(* PLC project Unnamed, Unknown Unnamed 1 *)
(* stored: creationDateTime 2026-08-16T23:05:33, modificationDateTime 2026-08-16T23:05:33 *)

FUNCTION_BLOCK CTU
  VAR_OUTPUT
    Q : BOOL;
    CV : INT;
  END_VAR
  VAR_INPUT
    CU : BOOL;
    R : BOOL;
    PV : INT;
  END_VAR

END_FUNCTION_BLOCK

FUNCTION_BLOCK F_TRIG
  VAR_OUTPUT
    Q : BOOL;
  END_VAR
  VAR_INPUT
    CLK : BOOL;
  END_VAR

END_FUNCTION_BLOCK

FUNCTION_BLOCK R_TRIG
  VAR_OUTPUT
    Q : BOOL;
  END_VAR
  VAR_INPUT
    CLK : BOOL;
  END_VAR

END_FUNCTION_BLOCK

FUNCTION_BLOCK SR
  VAR_OUTPUT
    Q1 : BOOL;
  END_VAR
  VAR_INPUT
    S1 : BOOL;
    R : BOOL;
  END_VAR

END_FUNCTION_BLOCK

FUNCTION_BLOCK TON
  VAR_OUTPUT
    Q : BOOL;
    ET : TIME;
  END_VAR
  VAR_INPUT
    IN : BOOL;
    PT : TIME;
  END_VAR

END_FUNCTION_BLOCK

PROGRAM main
  VAR
    Start_PB AT %QX1.0 : BOOL;  (* Simulated pushbutton, driven externally via Modbus coil *)
    Stop_PB AT %QX1.1 : BOOL;
    EStop_OK AT %QX1.2 : BOOL;
    Jam_Sensor AT %QX1.3 : BOOL;
    Part_Present AT %QX1.4 : BOOL;
    Reject_Sensor AT %QX1.5 : BOOL;
    Reset_PB AT %QX1.6 : BOOL;
    Conveyor_Motor AT %QX0.3 : BOOL;
    Fill_Actuator AT %QX0.4 : BOOL;
    Fault_Lamp AT %QX0.5 : BOOL;
    Reject_Gate AT %QX0.2 : BOOL;
    Machine_Running AT %QX0.0 : BOOL;
    Machine_Faulted AT %QX0.1 : BOOL;
    Cycle_Count AT %MW0 : INT;
    Good_Count AT %MW1 : INT;
    Reject_Count AT %MW2 : INT;
  END_VAR
  VAR
    SR0 : SR;
    R_TRIG0 : R_TRIG;
    Part_Edge : BOOL;
    CTU0 : CTU;
    TON0 : TON;
    CTU1 : CTU;
    CTU2 : CTU;
    TON1 : TON;
    F_TRIG0 : F_TRIG;
    Fault_Cleared : BOOL;
  END_VAR

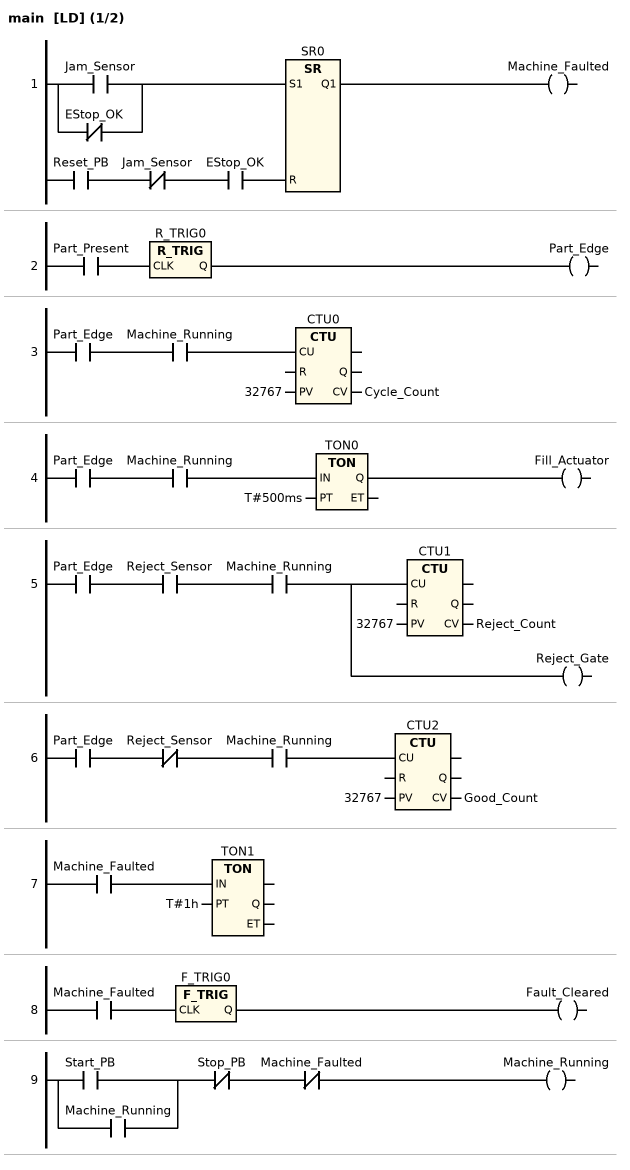
(* LD diagram, written out as Structured Text *)
Machine_Running := (Start_PB OR Machine_Running) AND NOT Stop_PB AND NOT Machine_Faulted;
SR0(S1 := Jam_Sensor OR NOT EStop_OK, R := Reset_PB AND NOT Jam_Sensor AND EStop_OK);
Machine_Faulted := SR0.Q1;
Conveyor_Motor := Machine_Running AND NOT Machine_Faulted;
Fault_Lamp := Machine_Faulted;
R_TRIG0(CLK := Part_Present);
Part_Edge := R_TRIG0.Q;
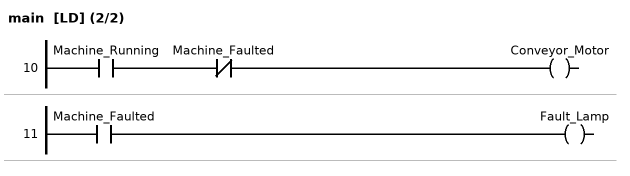
TON0(IN := Part_Edge AND Machine_Running, PT := T#500ms);
Fill_Actuator := TON0.Q;
Reject_Gate := Part_Edge AND Reject_Sensor AND Machine_Running;
F_TRIG0(CLK := Machine_Faulted);
Fault_Cleared := F_TRIG0.Q;
CTU0(CU := Part_Edge AND Machine_Running, R := , PV := 32767);
Cycle_Count := CTU0.CV;
 := TON0.ET;
CTU1(CU := Part_Edge AND Reject_Sensor AND Machine_Running, R := , PV := 32767);
Reject_Count := CTU1.CV;
CTU2(CU := Part_Edge AND NOT Reject_Sensor AND Machine_Running, R := , PV := 32767);
Good_Count := CTU2.CV;
TON1(IN := Machine_Faulted, PT := T#1h);
 := TON1.ET;
END_PROGRAM

CONFIGURATION Config0
  RESOURCE Res0 ON PLC
    TASK task0(INTERVAL := T#100ms, PRIORITY := 1);
    PROGRAM instance0 WITH task0 : main;
  END_RESOURCE
END_CONFIGURATION
